Fanuc TP program (LS listing): UP100.LS

/PROG  UP100
/ATTR
OWNER		= MNEDITOR;
COMMENT		= "";
PROG_SIZE	= 187;
CREATE		= DATE 24-04-14  TIME 11:05:32;
MODIFIED	= DATE 24-04-14  TIME 11:06:12;
FILE_NAME	= ;
VERSION		= 0;
LINE_COUNT	= 2;
MEMORY_SIZE	= 551;
PROTECT		= READ_WRITE;
TCD:  STACK_SIZE	= 0,
      TASK_PRIORITY	= 50,
      TIME_SLICE	= 0,
      BUSY_LAMP_OFF	= 0,
      ABORT_REQUEST	= 0,
      PAUSE_REQUEST	= 0;
DEFAULT_GROUP	= 1,1,1,1,*;
CONTROL_CODE	= 00000000 00000000;
/APPL

CORNER_SPEED_HEADER;
  ENABLE_CORNER_SPEED   : FALSE;
/MN
   1:  UFRAME_NUM=0 ;
   2:  UTOOL_NUM=0 ;
/POS
/END
